DATA_BLOCK "dbPlcHmiMTR"
{ S7_Optimized_Access := 'FALSE' }
VERSION : 0.1
 STRUCT
   MTR : Array[2000..2011] of "UDT_CM_MTR_N";
 END_STRUCT;

BEGIN
END_DATA_BLOCK
